FUNCTION_BLOCK Msg3002_NavitrolStatus EXTENDS TcpIpCommandResultFilter IMPLEMENTS I_Navitrol_Status
VAR
	CycleTime		  : TIME := T#100MS; //maximum interval 1 second
	Timer			  : TON;
	Command			  : ST_TcpIpPayload;
	ReceiveBuffer	  : U_Recived_bytes_from_Navitrol;
	Supervisor_Status : ST_3002_Supervisor_Status;
	Navitrol_status	  : ST_3102_Navitrol_status;
END_VAR

METHOD CyclicLogic
SUPER^.CyclicLogic();
Timer(IN := NOT Timer.Q, PT := CycleTime);
IF Timer.Q AND TcpIpConnection.ConnectionState = eSOCKET_CONNECTED THEN
	F_SetHeaderInfo(Supervisor_Status);
	F_SetSectionHeaderInfo(Supervisor_Status.Manual_section);
	F_SetSectionHeaderInfo(Supervisor_Status.Battery_section);
	MEMSET(ADR(Command), 0, SIZEOF(Command));
	Command.Size := SIZEOF(Supervisor_Status);
	MEMCPY(ADR(Command.Data), ADR(Supervisor_Status), Command.Size);
	TcpIpConnection.SendCommand(ADR(Command));
	CommandActive := TRUE;
END_IF
END_METHOD

PROPERTY NavitrolStatus : REFERENCE TO ST_3102_Navitrol_status
GET
NavitrolStatus REF= Navitrol_status;
END_GET
END_PROPERTY

PROPERTY SupervisorStatus : REFERENCE TO ST_3002_Supervisor_Status
GET
SupervisorStatus REF= Supervisor_Status;
END_GET
END_PROPERTY

METHOD UpdateCommandResult
VAR_INPUT
	Response : POINTER TO ST_TcpIpPayload;
END_VAR

VAR_INST
	ReceiveCounter : UDINT;
END_VAR
MEMCPY(ADR(ReceiveBuffer), ADR(Response^.Data), SIZEOF(ReceiveBuffer));
IF ReceiveBuffer.Header.Message_ID = 3102 THEN
	ReceiveCounter := ReceiveCounter + 1;
	MEMCPY(destAddr := ADR(Navitrol_status), srcAddr := ADR(ReceiveBuffer), n := SIZEOF(Navitrol_status));
	CommandActive := FALSE;
END_IF
END_METHOD

END_FUNCTION_BLOCK

(* stored: Version 1.1.0.1
   POU Msg3002_NavitrolStatus: Id {0ad2d1b3-a026-4051-b631-30c9c5f84423}, SpecialFunc None
   Method CyclicLogic: Id {38ed6b6e-d9ff-411d-aef6-4aea099e5bc6}
   Property NavitrolStatus: Id {f380a5dd-a7fc-41d6-8523-e946e6423408}
   Get Get: Id {63fc1aa6-8e88-4b9a-8c46-1b42d35b1154}
   Property SupervisorStatus: Id {d364014a-7ad2-4251-8cdb-edbd948ae274}
   Get Get: Id {660a7054-ae99-4766-b466-b16c92ccff9b}
   Method UpdateCommandResult: Id {1a4e6bd8-e8a3-4831-8629-4db1d87295eb} *)
